PROGRAM PRG_Compilation
VAR
END_VAR

END_PROGRAM

(* stored: Version 1.1.0.1
   POU PRG_Compilation: Id {467eb2b3-ada0-4736-a305-ff78f2de95cf}, SpecialFunc None *)
